TYPE ST_Station_HMI :
STRUCT
	iStep			:UINT;
	bInterlocksOK	:BOOL;
	bReset			:BOOL;
	iStatus			:UINT;
END_STRUCT
END_TYPE

(* stored: Version 1.1.0.1
   DUT ST_Station_HMI: Id {afa8b352-23ca-411a-88f0-c51e8f2209d8} *)
